// TwinCAT 3 PLC project AdsGamepad
// Title: AdsGamepad
// Company: Beckhoff Community
// Author: Beckhoff USA Community
// ProjectVersion: 2.3.0
// Description: A library to communicate with the ADS Gamepad Service
// ProgramVersion: 3.1.4026.24
// libraries:
//   Tc2_System, * (Beckhoff Automation GmbH)
//   Tc3_Module, * (Beckhoff Automation GmbH)
// project tree:
//   DUTs/ E_Gamepad_Battery_Levels.TcDUT, E_Gamepad_Battery_Types.TcDUT, E_Gamepad_Handshake_State.TcDUT, ST_Gamepad_ADS_Inputs.TcDUT, ST_Gamepad_Ext_ADS_Inputs.TcDUT, ST_Gamepad_Ext_Battery.TcDUT, ST_Gamepad_Ext_Buttons.TcDUT, ST_Gamepad_Motion.TcDUT, ST_Gamepad_Touch_Point.TcDUT, ST_Gamepad_Touchpad.TcDUT, ST_Gamepad_Buttons.TcDUT, ST_Gamepad_Command_Status.TcDUT, ST_Gamepad_DPad.TcDUT, ST_Gamepad_Joystick.TcDUT, ST_Gamepad_Rumble.TcDUT, ST_Gamepad_Service_Info.TcDUT, ST_Gamepad_Status.TcDUT
//   DUTs/LowerLevel/ ST_Gamepad_Buttons_Bits.TcDUT, ST_Gamepad_Ext_Touch_Raw.TcDUT, ST_Gamepad_State_Bits.TcDUT
//   FBs/ FB_Gamepad_Controller.TcPOU
//   Project Information/ F_GetCompany.TcPOU (not stored), F_GetTitle.TcPOU, F_GetVersion.TcPOU
//   Version/ Global_Version.TcGVL

// ---- DUTs/E_Gamepad_Battery_Levels.TcDUT
{attribute 'qualified_only'}
{attribute 'strict'}
TYPE E_Gamepad_Battery_Levels :
(
	// Battery is Empty or Unknown
	Empty := 0,
	// Battery is at low level
	Low := 1,
	// Battery is at medium level
	Medium := 2,
	// Battery is at full level
	Full := 3
);
END_TYPE

// ---- DUTs/E_Gamepad_Battery_Types.TcDUT
{attribute 'qualified_only'}
{attribute 'strict'}
TYPE E_Gamepad_Battery_Types :
(
	// Battery is disconnected
	Disconnected := 0,
	// Battery is wired
	Wired := 1,
	// Battery is alkaline
	Alkaline := 2,
	// Battery is NiMH
	NIMH := 3,
	// Battery is unknown
	Unknown := 4
);
END_TYPE

// ---- DUTs/E_Gamepad_Handshake_State.TcDUT
{attribute 'qualified_only'}
{attribute 'strict'}
TYPE E_Gamepad_Handshake_State :
(
	// No handshake attempt has run yet
	NotStarted := 0,
	// The read of the service info block is in flight
	Busy := 1,
	// The service answered and the contract versions are compatible
	Compatible := 2,
	// The last attempt got no answer. The service predates the info block or was not
	// reachable yet; the handshake keeps retrying. Data exchange still works
	Unsupported := 3,
	// The service speaks a newer contract major version. Check for a library update
	Mismatch := 4
);
END_TYPE

// ---- DUTs/LowerLevel/ST_Gamepad_Buttons_Bits.TcDUT
TYPE ST_Gamepad_Buttons_Bits :
STRUCT
	xDPAD_UP  			: BIT;
    xDPAD_DOWN  		: BIT;
    xDPAD_LEFT  		: BIT;
    xDPAD_RIGHT  		: BIT;
    xSTART  			: BIT;
    xBACK  				: BIT;
    xLEFT_THUMB  		: BIT;
    xRIGHT_THUMB  		: BIT;   
	xLEFT_SHOULDER  	: BIT;
    xRIGHT_SHOULDER  	: BIT;
	{attribute 'hide'}
	xFiller1 			: BIT;
	{attribute 'hide'}
	xFiller2			: BIT;
	xA  				: BIT;
	xB  				: BIT;
	xX  				: BIT;
	xY  				: BIT;
END_STRUCT
END_TYPE

// ---- DUTs/LowerLevel/ST_Gamepad_Ext_Touch_Raw.TcDUT
// One touchpad contact exactly as it arrives in the extended block.
// Use the P_Touchpad property for the friendly form. Layout is frozen.
{attribute 'pack_mode' := '4'}
TYPE ST_Gamepad_Ext_Touch_Raw :
STRUCT
	// 1 while a finger is on the pad, 0 otherwise
	nActive		: USINT;
	// Counts contacts, so a new touch gets a new number
	nContactId	: USINT;
	// Position across the pad, 0 to 1919
	nX			: UINT;
	// Position down the pad, 0 to 1079
	nY			: UINT;
END_STRUCT
END_TYPE

// ---- DUTs/LowerLevel/ST_Gamepad_State_Bits.TcDUT
TYPE ST_Gamepad_State_Bits :
STRUCT
	xConnected  				: BIT;
	xBattery_Type_Disconnected	: BIT;
	xBattery_Type_Wired			: BIT;
	xBattery_Type_Alkaline		: BIT;
	xBattery_Type_NIMH			: BIT;
	xBattery_Type_Unknown		: BIT;
	xBattery_Level_Empty		: BIT;
	xBattery_Level_Low			: BIT;
	xBattery_Level_Medium		: BIT;
	xBattery_Level_Full			: BIT;
	
	{attribute 'hide'}
	xFiller10					: BIT;
	{attribute 'hide'}
	xFiller11					: BIT;
	{attribute 'hide'}
	xFiller12					: BIT;
	{attribute 'hide'}
	xFiller13					: BIT;
	{attribute 'hide'}
	xFiller14					: BIT;
	{attribute 'hide'}
	xFiller15					: BIT;
END_STRUCT
END_TYPE

// ---- DUTs/ST_Gamepad_ADS_Inputs.TcDUT
TYPE ST_Gamepad_ADS_Inputs :
STRUCT
	// Controller Number
	iControllerNumber	: INT;
	// Struct of Left Joystick values
	stLeft_Joystick 	: ST_Gamepad_Joystick;
	// Struct of Right Joystick values
	stRight_Joystick 	: ST_Gamepad_Joystick;
	// Left Trigger value
	fLeft_Trigger 		: REAL;
	// Right Trigger value
	fRight_Trigger 		: REAL;
	// Struct of individual raw button bits read from the controller
	bButtons 			: ST_Gamepad_Buttons_Bits;
	// Struct of individual raw status bits read from the controller
	bStatus				: ST_Gamepad_State_Bits;
END_STRUCT
END_TYPE

// ---- DUTs/ST_Gamepad_Ext_ADS_Inputs.TcDUT
// Mirror of the 96 byte extended block served per controller since wire
// contract 1.3. Older services answer the read with an error and the
// struct then reads all zero. A slot without extended data, for example
// an Xbox controller, reads all zero with the present flag clear.
// Layout is frozen.
{attribute 'pack_mode' := '4'}
TYPE ST_Gamepad_Ext_ADS_Inputs :
STRUCT
	// Size of the block, 96 when the service serves it
	nExtSize			: UINT;
	// Layout version of the fields below, 1 today
	nExtLayoutVersion	: UINT;
	// Bit 0 PS, bit 1 Mute, bit 2 touchpad click
	nExtButtons			: WORD;
	// Bit 0 set means this slot supplies extended data right now.
	// Bit 1 set means the battery fields below hold data, since contract 1.4
	nExtFlags			: WORD;
	// Raw motion sensor values. Interpreting them is application code
	nGyroX				: INT;
	nGyroY				: INT;
	nGyroZ				: INT;
	nAccelX				: INT;
	nAccelY				: INT;
	nAccelZ				: INT;
	// Up to two touchpad contacts
	stTouch0			: ST_Gamepad_Ext_Touch_Raw;
	stTouch1			: ST_Gamepad_Ext_Touch_Raw;
	// Report counter from the pad, widened by the service. A value that
	// keeps moving proves the input stream is alive
	nSequence			: UDINT;
	// Battery data since contract 1.4, gated on flag bit 1: charge in
	// percent, then bit 0 charging and bit 1 full. Use P_Ext_Battery
	nBatteryPercent		: USINT;
	nBatteryFlags		: USINT;
	nReserved			: UINT;
	// Reserved for future contract versions, always zero today
	aReserved			: ARRAY [0..55] OF BYTE;
END_STRUCT
END_TYPE

// ---- DUTs/ST_Gamepad_Ext_Battery.TcDUT
// Battery state from the extended block. Valid only while bValid is TRUE:
// a service older than 2.6.0 does not serve it, an Xbox slot has none, and
// a pad error state reads as not valid rather than as a guess.
TYPE ST_Gamepad_Ext_Battery :
STRUCT
	// TRUE while the service supplies battery data for this slot
	bValid		: BOOL;
	// Charge from 0 to 100 percent
	nPercent	: USINT;
	// TRUE while the pad charges over its cable
	bCharging	: BOOL;
	// TRUE when the battery is full
	bFull		: BOOL;
END_STRUCT
END_TYPE

// ---- DUTs/ST_Gamepad_Ext_Buttons.TcDUT
// Buttons beyond the classic gamepad surface. A PlayStation pad supplies
// them through the extended block; on other pads they stay FALSE.
TYPE ST_Gamepad_Ext_Buttons :
STRUCT
	// The PS logo button
	bPS				: BOOL;
	// The microphone mute button
	bMute			: BOOL;
	// The touchpad pressed as a button
	bTouchpad_Click	: BOOL;
END_STRUCT
END_TYPE

// ---- DUTs/ST_Gamepad_Motion.TcDUT
// Raw motion sensor values from the pad. The units are the sensor's own;
// interpreting or filtering them is application code. At rest the gyro
// values show small noise and the accelerometer shows gravity.
TYPE ST_Gamepad_Motion :
STRUCT
	nGyroX	: INT;
	nGyroY	: INT;
	nGyroZ	: INT;
	nAccelX	: INT;
	nAccelY	: INT;
	nAccelZ	: INT;
END_STRUCT
END_TYPE

// ---- DUTs/ST_Gamepad_Touch_Point.TcDUT
// One finger on the touchpad in friendly form.
TYPE ST_Gamepad_Touch_Point :
STRUCT
	// TRUE while the finger touches the pad
	bActive		: BOOL;
	// Counts contacts, so a new touch gets a new number
	nContactId	: USINT;
	// Position across the pad, 0 to 1919
	nX			: UINT;
	// Position down the pad, 0 to 1079
	nY			: UINT;
END_STRUCT
END_TYPE

// ---- DUTs/ST_Gamepad_Touchpad.TcDUT
// The touchpad with its two possible contacts.
TYPE ST_Gamepad_Touchpad :
STRUCT
	stPoint1	: ST_Gamepad_Touch_Point;
	stPoint2	: ST_Gamepad_Touch_Point;
END_STRUCT
END_TYPE

// ---- DUTs/ST_Gamepad_Buttons.TcDUT
TYPE ST_Gamepad_Buttons :
STRUCT
	// Directional Pad Struct
	DPad				: ST_Gamepad_DPad;
	// Start Button
    bStart  			: BOOL;
	// Back Button
    bBack  				: BOOL;
	// Pressing in the Left Thumbstick
    bLeft_Thumbstick  	: BOOL;
	// Pressing in the Right Thumbstick
    bRight_Thumbstick  	: BOOL;
	// Left Shoulder Button  
	bLeft_Shoulder  	: BOOL;
	// Right Shoulder Button
    bRight_Shoulder  	: BOOL;
	// Button A
	bA_Button  			: BOOL;
	// Button B
	bB_Button  			: BOOL;
	// Button X
	bX_Button  			: BOOL;
	// Button Y
	bY_Button  			: BOOL;
END_STRUCT
END_TYPE

// ---- DUTs/ST_Gamepad_Command_Status.TcDUT
TYPE ST_Gamepad_Command_Status :
STRUCT
	// Command has been completed
	bDone 	: BOOL;
	// Command is busy
	bBusy 	: BOOL;
	// Command has an error
	bError 	: BOOL;
END_STRUCT
END_TYPE

// ---- DUTs/ST_Gamepad_DPad.TcDUT
TYPE ST_Gamepad_DPad :
STRUCT
	// Up Button on DPad
	bUp  		: BOOL;
	// Down Button on DPad
    bDown  		: BOOL;
	// Left Button on DPad
    bLeft  		: BOOL;
	// Right Button on DPad
    bRight  	: BOOL;
END_STRUCT
END_TYPE

// ---- DUTs/ST_Gamepad_Joystick.TcDUT
TYPE ST_Gamepad_Joystick :
STRUCT
	// Joystick's X Value (-100...100%)
	fX : REAL;
	// Joystick's Y Value (-100...100%)
	fY : REAL;
END_STRUCT
END_TYPE

// ---- DUTs/ST_Gamepad_Rumble.TcDUT
TYPE ST_Gamepad_Rumble :
STRUCT
	// Rumble of left motor (0..100%)
	fLeftMotor 	: REAL;
	// Rumble of right motor (0..100%)
	fRightMotor : REAL;
END_STRUCT
END_TYPE

// ---- DUTs/ST_Gamepad_Service_Info.TcDUT
// Mirror of the 32 byte service info block served at IndexGroup 16#F000.
// Services older than 2.1.0 do not serve this block. Layout is frozen.
TYPE ST_Gamepad_Service_Info :
STRUCT
	// Wire contract version the service speaks. This library expects major 1
	nContractMajor	: UINT;
	nContractMinor	: UINT;
	// Version of the running service program
	nServiceMajor	: UINT;
	nServiceMinor	: UINT;
	nServicePatch	: UINT;
	nReserved		: UINT;
	// Capability bits. Bit 0 means the XInput backend is present
	dwCapabilities	: UDINT;
	// Reserved for future contract versions, always zero today
	aReserved		: ARRAY [0..15] OF BYTE;
END_STRUCT
END_TYPE

// ---- DUTs/ST_Gamepad_Status.TcDUT
TYPE ST_Gamepad_Status :
STRUCT
	// Controller's ID
	iControllerNumber  	: INT;
	// Controller is connected to the PC
	bConnected  		: BOOL;
	// Controller is disconnected from the PC
	bDisconnected  		: BOOL;
	// Battery Type
	eBattery_Type 		: E_Gamepad_Battery_Types;
	// Battery Level
	eBattery_Level 		: E_Gamepad_Battery_Levels;
END_STRUCT
END_TYPE

// ---- Version/Global_Version.TcGVL
{attribute 'TcGenerated'}
{attribute 'no-analysis'}
{attribute 'linkalways'}
// This function has been automatically generated from the project information.
VAR_GLOBAL CONSTANT
	{attribute 'const_non_replaced'}
	stLibVersion_AdsGamepad : ST_LibVersion := (iMajor := 2, iMinor := 3, iBuild := 0, iRevision := 0, nFlags := 1, sVersion := '2.3.0');
END_VAR

// ---- FBs/FB_Gamepad_Controller.TcPOU
{attribute 'no_explicit_call' := 'do not call this FB directly, call Cycle instead'} 
FUNCTION_BLOCK FB_Gamepad_Controller
VAR
	{attribute 'hide'}
	_AmsNetId : T_AMSNETID;
	{attribute 'hide'}
	_WriteServerData : ADSWRITE;
	{attribute 'hide'}
	_ReadServerData : ADSREAD;
	// RAW ADS Inputs for debug (Use properties to access items)
	stGamepadInputs : ST_Gamepad_ADS_Inputs;
	{attribute 'hide'}
	_stRumble : ST_Gamepad_Rumble;
	{attribute 'hide'}
	_IDXGRP : UDINT;
	{attribute 'hide'}
	_rumbleCommand 			: ST_Gamepad_Command_Status;
	{attribute 'hide'}
	_stControllerButtons 	: ST_Gamepad_Buttons;
	{attribute 'hide'}
	_stControllerStatus		: ST_Gamepad_Status;
	{attribute 'hide'}
	_stLeftJoystick 		: ST_Gamepad_Joystick;
	{attribute 'hide'}
	_stRightJoystick 		: ST_Gamepad_Joystick;
	{attribute 'hide'}
	_fLeftTrigger 			: REAL;
	{attribute 'hide'}
	_fRightTrigger 			: REAL;
	{attribute 'hide'}
	_bSetRumbleEvent 		: BOOL; // Internal indication of an ADS write event
	{attribute 'hide'}
	_bSetRumbleEventLogged	: BOOL; // Check if the Set Rumble event is being called too many times
	{attribute 'hide'}
	_ReadServiceInfo : ADSREAD;
	{attribute 'hide'}
	_stServiceInfo : ST_Gamepad_Service_Info;
	{attribute 'hide'}
	_eHandshakeState : E_Gamepad_Handshake_State;
	{attribute 'hide'}
	_nHandshakeRetryCycles : UDINT; // Counts cycles between handshake retries after a failed attempt
	{attribute 'hide'}
	_ReadExtData : ADSREAD;
	// RAW extended block for debug (Use properties to access items)
	stGamepadExtInputs : ST_Gamepad_Ext_ADS_Inputs;
	{attribute 'hide'}
	_stExtButtons : ST_Gamepad_Ext_Buttons;
	{attribute 'hide'}
	_stTouchpad : ST_Gamepad_Touchpad;
	{attribute 'hide'}
	_stMotion : ST_Gamepad_Motion;
	{attribute 'hide'}
	_stExtBattery : ST_Gamepad_Ext_Battery;
END_VAR

// This method is called cyclically to update the controller inputs
METHOD Cycle : BOOL
// Read the current inputs
THIS^._ReadServerData(
	NETID:= THIS^._AmsNetId, 
	PORT:= 25733, 
	IDXGRP:= THIS^._IDXGRP, 
	IDXOFFS:= 0, 
	LEN:= SIZEOF(THIS^.stGamepadInputs), 
	DESTADDR:= ADR(THIS^.stGamepadInputs), 
	READ:= TRUE, 
	TMOUT:= T#5S,
	ERR=>);
	
// If there is an error in reading from the server, shut all inputs off
IF THIS^._ReadServerData.ERR THEN
	memset(ADR(THIS^.stGamepadInputs), 0, SIZEOF(THIS^.stGamepadInputs));
END_IF

// Stop read command
THIS^._ReadServerData(
	NETID:= THIS^._AmsNetId, 
	PORT:= 25733, 
	IDXGRP:= THIS^._IDXGRP, 
	IDXOFFS:= 0, 
	LEN:= SIZEOF(THIS^.stGamepadInputs), 
	DESTADDR:= ADR(THIS^.stGamepadInputs), 
	READ:= FALSE, 
	TMOUT:= T#5S,
	ERR=>);
	

// Handle any write requests for the rumble
// Write the new values
THIS^._WriteServerData(
	NETID:= THIS^._AmsNetId, 
	PORT:= 25733, 
	IDXGRP:= THIS^._IDXGRP, 
	IDXOFFS:= 16, 
	LEN:= SIZEOF(THIS^._stRumble), 
	SRCADDR:= ADR(THIS^._stRumble), 
	WRITE:= THIS^._bSetRumbleEvent, 
	TMOUT:= T#5S);
	
// Update the status of the current command if active
IF 	THIS^._bSetRumbleEvent THEN
	THIS^.P_SetRumble.bBusy := THIS^._WriteServerData.BUSY;
	THIS^.P_SetRumble.bError := THIS^._WriteServerData.ERR;
END_IF

// Check if it's done writing
IF THIS^._bSetRumbleEvent AND NOT THIS^._WriteServerData.BUSY THEN
	IF NOT THIS^._WriteServerData.ERR THEN
		THIS^.P_SetRumble.bDone := TRUE;
	END_IF
	// Turn off the write request
	THIS^._WriteServerData(
		NETID:= THIS^._AmsNetId, 
		PORT:= 25733, 
		IDXGRP:= THIS^._IDXGRP, 
		IDXOFFS:= 16, 
		LEN:= SIZEOF(THIS^._stRumble), 
		SRCADDR:= ADR(THIS^._stRumble), 
		WRITE:= FALSE, 
		TMOUT:= T#5S);

	THIS^._bSetRumbleEvent := FALSE;
END_IF

// Version handshake against the service info block at IndexGroup 16#F000.
// Services older than 2.1.0 answer with an error, which is fine. Data exchange works either way.
// A failed attempt reports Unsupported and retries in the background, so a service that starts
// after the PLC, for example right after an install, still gets a handshake without a PLC restart
CASE THIS^._eHandshakeState OF
	E_Gamepad_Handshake_State.NotStarted:
		THIS^._ReadServiceInfo(
			NETID:= THIS^._AmsNetId,
			PORT:= 25733,
			IDXGRP:= 16#F000,
			IDXOFFS:= 0,
			LEN:= SIZEOF(THIS^._stServiceInfo),
			DESTADDR:= ADR(THIS^._stServiceInfo),
			READ:= TRUE,
			TMOUT:= T#5S);
		THIS^._eHandshakeState := E_Gamepad_Handshake_State.Busy;

	E_Gamepad_Handshake_State.Busy:
		THIS^._ReadServiceInfo(READ:= TRUE);
		IF THIS^._ReadServiceInfo.ERR THEN
			// No answer. The service predates version 2.1.0 or it was not reachable, for example
			// while it was still starting. The Unsupported case below retries later
			memset(ADR(THIS^._stServiceInfo), 0, SIZEOF(THIS^._stServiceInfo));
			THIS^._eHandshakeState := E_Gamepad_Handshake_State.Unsupported;
			THIS^._ReadServiceInfo(READ:= FALSE);
		ELSIF NOT THIS^._ReadServiceInfo.BUSY THEN
			IF THIS^._stServiceInfo.nContractMajor = 1 THEN
				THIS^._eHandshakeState := E_Gamepad_Handshake_State.Compatible;
			ELSE
				ADSLOGSTR( msgCtrlMask := ADSLOG_MSGTYPE_WARN, msgFmtStr := 'PLC Msg.: The ADS Gamepad Service speaks a newer wire contract, update the AdsGamepad library: %s', strArg := 'FB_Gamepad_Controller');
				THIS^._eHandshakeState := E_Gamepad_Handshake_State.Mismatch;
			END_IF
			THIS^._ReadServiceInfo(READ:= FALSE);
		END_IF

	E_Gamepad_Handshake_State.Unsupported:
		// Retry the handshake in the background without leaving the reported state,
		// so consumers watching P_Handshake_State never see it flap. A genuinely old
		// service answers every retry with an error and the state simply stays
		// Unsupported; a service that was only starting late answers and the state
		// moves on. 5000 cycles is five seconds at a one millisecond PLC cycle
		THIS^._nHandshakeRetryCycles := THIS^._nHandshakeRetryCycles + 1;
		IF THIS^._nHandshakeRetryCycles >= 5000 THEN
			THIS^._ReadServiceInfo(
				NETID:= THIS^._AmsNetId,
				PORT:= 25733,
				IDXGRP:= 16#F000,
				IDXOFFS:= 0,
				LEN:= SIZEOF(THIS^._stServiceInfo),
				DESTADDR:= ADR(THIS^._stServiceInfo),
				READ:= TRUE,
				TMOUT:= T#5S);
			IF THIS^._ReadServiceInfo.ERR THEN
				// Still no answer; reset the read and count up to the next attempt
				memset(ADR(THIS^._stServiceInfo), 0, SIZEOF(THIS^._stServiceInfo));
				THIS^._ReadServiceInfo(READ:= FALSE);
				THIS^._nHandshakeRetryCycles := 0;
			ELSIF NOT THIS^._ReadServiceInfo.BUSY THEN
				IF THIS^._stServiceInfo.nContractMajor = 1 THEN
					THIS^._eHandshakeState := E_Gamepad_Handshake_State.Compatible;
				ELSE
					ADSLOGSTR( msgCtrlMask := ADSLOG_MSGTYPE_WARN, msgFmtStr := 'PLC Msg.: The ADS Gamepad Service speaks a newer wire contract, update the AdsGamepad library: %s', strArg := 'FB_Gamepad_Controller');
					THIS^._eHandshakeState := E_Gamepad_Handshake_State.Mismatch;
				END_IF
				THIS^._ReadServiceInfo(READ:= FALSE);
				THIS^._nHandshakeRetryCycles := 0;
			END_IF
		END_IF
END_CASE
END_METHOD

METHOD FB_init : BOOL
VAR_INPUT
	bInitRetains : BOOL; // if TRUE, the retain variables are initialized (warm start / cold start)
	bInCopyCode : BOOL;  // if TRUE, the instance afterwards gets moved into the copy code (online change)
	NetID 				: T_AMSNETID := ''; // AMS Net ID of the ADS Gamepad Service
	iControllerNumber 	: UINT(1..4) := 1; // The controller number for the controller you'd like to use
END_VAR
THIS^._AmsNetId := NetID;
THIS^._IDXGRP := iControllerNumber * 16#10000;
END_METHOD

{attribute 'monitoring':='call'}
// Structure of the different active buttons
PROPERTY P_Buttons : REFERENCE TO ST_Gamepad_Buttons
GET
IF THIS^.stGamepadInputs.bStatus.xConnected THEN	
	THIS^._stControllerButtons.DPad.bUp				:= THIS^.stGamepadInputs.bButtons.xDPAD_UP;
	THIS^._stControllerButtons.DPad.bDown			:= THIS^.stGamepadInputs.bButtons.xDPAD_DOWN;
	THIS^._stControllerButtons.DPad.bLeft			:= THIS^.stGamepadInputs.bButtons.xDPAD_LEFT;
	THIS^._stControllerButtons.DPad.bRight			:= THIS^.stGamepadInputs.bButtons.xDPAD_RIGHT;
	THIS^._stControllerButtons.bStart  				:= THIS^.stGamepadInputs.bButtons.xSTART;
	THIS^._stControllerButtons.bBack  				:= THIS^.stGamepadInputs.bButtons.xBACK;
	THIS^._stControllerButtons.bLeft_Thumbstick  	:= THIS^.stGamepadInputs.bButtons.xLEFT_THUMB;
	THIS^._stControllerButtons.bRight_Thumbstick 	:= THIS^.stGamepadInputs.bButtons.xRIGHT_THUMB;
	THIS^._stControllerButtons.bLeft_Shoulder  		:= THIS^.stGamepadInputs.bButtons.xLEFT_SHOULDER;
	THIS^._stControllerButtons.bRight_Shoulder  	:= THIS^.stGamepadInputs.bButtons.xRIGHT_SHOULDER;
	THIS^._stControllerButtons.bA_Button  			:= THIS^.stGamepadInputs.bButtons.xA;
	THIS^._stControllerButtons.bB_Button  			:= THIS^.stGamepadInputs.bButtons.xB;
	THIS^._stControllerButtons.bX_Button  			:= THIS^.stGamepadInputs.bButtons.xX;
	THIS^._stControllerButtons.bY_Button  			:= THIS^.stGamepadInputs.bButtons.xY;
ELSE
	THIS^._stControllerButtons.DPad.bUp				:= FALSE;
	THIS^._stControllerButtons.DPad.bDown			:= FALSE;
	THIS^._stControllerButtons.DPad.bLeft			:= FALSE;
	THIS^._stControllerButtons.DPad.bRight			:= FALSE;
	THIS^._stControllerButtons.bStart  				:= FALSE;
	THIS^._stControllerButtons.bBack  				:= FALSE;
	THIS^._stControllerButtons.bLeft_Thumbstick  	:= FALSE;
	THIS^._stControllerButtons.bRight_Thumbstick 	:= FALSE;
	THIS^._stControllerButtons.bLeft_Shoulder  		:= FALSE;
	THIS^._stControllerButtons.bRight_Shoulder  	:= FALSE;
	THIS^._stControllerButtons.bA_Button  			:= FALSE;
	THIS^._stControllerButtons.bB_Button  			:= FALSE;
	THIS^._stControllerButtons.bX_Button  			:= FALSE;
	THIS^._stControllerButtons.bY_Button  			:= FALSE;
END_IF
P_Buttons REF= THIS^._stControllerButtons;
END_GET
END_PROPERTY

{attribute 'monitoring':='call'}
// Returns a structure of data for the XY Joystick values
PROPERTY P_Left_Joystick : REFERENCE TO ST_Gamepad_Joystick
GET
IF THIS^.stGamepadInputs.bStatus.xConnected THEN	
	THIS^._stLeftJoystick.fX := THIS^.stGamepadInputs.stLeft_Joystick.fX;
	THIS^._stLeftJoystick.fY := THIS^.stGamepadInputs.stLeft_Joystick.fY;
ELSE
	THIS^._stLeftJoystick.fX := 0;
	THIS^._stLeftJoystick.fY := 0;
END_IF
P_Left_Joystick REF= THIS^._stLeftJoystick;
END_GET
END_PROPERTY

{attribute 'monitoring':='call'}
// Left trigger value
PROPERTY P_Left_Trigger : REFERENCE TO REAL
GET
IF THIS^.stGamepadInputs.bStatus.xConnected THEN	
	THIS^._fLeftTrigger := THIS^.stGamepadInputs.fLeft_Trigger;
ELSE
	THIS^._fLeftTrigger := 0;
END_IF
P_Left_Trigger REF= THIS^._fLeftTrigger;
END_GET
END_PROPERTY

{attribute 'monitoring':='call'}
// Returns a structure of data for the XY Joystick values
PROPERTY P_Right_Joystick : REFERENCE TO ST_Gamepad_Joystick
GET
IF THIS^.stGamepadInputs.bStatus.xConnected THEN	
	THIS^._stRightJoystick.fX := THIS^.stGamepadInputs.stRight_Joystick.fX;
	THIS^._stRightJoystick.fY := THIS^.stGamepadInputs.stRight_Joystick.fY;
ELSE
	THIS^._stRightJoystick.fX := 0;
	THIS^._stRightJoystick.fY := 0;
END_IF
P_Right_Joystick REF= THIS^._stRightJoystick;
END_GET
END_PROPERTY

{attribute 'monitoring':='call'}
// Right trigger value
PROPERTY P_Right_Trigger : REFERENCE TO REAL
GET
IF THIS^.stGamepadInputs.bStatus.xConnected THEN	
	THIS^._fRightTrigger := THIS^.stGamepadInputs.fRight_Trigger;
ELSE
	THIS^._fRightTrigger := 0;
END_IF
P_Right_Trigger REF= THIS^._fRightTrigger;
END_GET
END_PROPERTY

{attribute 'monitoring':='call'}
// Status of the SetRumble method
PROPERTY P_SetRumble : REFERENCE TO ST_Gamepad_Command_Status
GET
P_SetRumble REF= THIS^._rumbleCommand;
END_GET
END_PROPERTY

{attribute 'monitoring':='call'}
// Structure of the controller capabilites and status
PROPERTY P_Status : REFERENCE TO ST_Gamepad_Status
GET
IF THIS^.stGamepadInputs.bStatus.xConnected THEN	
	THIS^._stControllerStatus.bConnected 		:= TRUE;
	THIS^._stControllerStatus.bDisconnected 	:= FALSE;
	THIS^._stControllerStatus.iControllerNumber := THIS^.stGamepadInputs.iControllerNumber;
ELSE
	THIS^._stControllerStatus.bConnected 		:= FALSE;
	THIS^._stControllerStatus.bDisconnected 	:= TRUE;
	THIS^._stControllerStatus.iControllerNumber := 0;
END_IF

IF THIS^.stGamepadInputs.bStatus.xBattery_Type_Disconnected THEN
	THIS^._stControllerStatus.eBattery_Type := E_Gamepad_Battery_Types.Disconnected;
END_IF

IF THIS^.stGamepadInputs.bStatus.xBattery_Type_Wired THEN
	THIS^._stControllerStatus.eBattery_Type := E_Gamepad_Battery_Types.Wired;
END_IF

IF THIS^.stGamepadInputs.bStatus.xBattery_Type_Alkaline THEN
	THIS^._stControllerStatus.eBattery_Type := E_Gamepad_Battery_Types.Alkaline;
END_IF

IF THIS^.stGamepadInputs.bStatus.xBattery_Type_NIMH THEN
	THIS^._stControllerStatus.eBattery_Type := E_Gamepad_Battery_Types.NIMH;
END_IF

IF THIS^.stGamepadInputs.bStatus.xBattery_Type_Unknown THEN
	THIS^._stControllerStatus.eBattery_Type := E_Gamepad_Battery_Types.Unknown;
END_IF

IF THIS^.stGamepadInputs.bStatus.xBattery_Level_Empty THEN
	THIS^._stControllerStatus.eBattery_Level := E_Gamepad_Battery_Levels.Empty;
END_IF

IF THIS^.stGamepadInputs.bStatus.xBattery_Level_Low THEN
	THIS^._stControllerStatus.eBattery_Level := E_Gamepad_Battery_Levels.Low;
END_IF

IF THIS^.stGamepadInputs.bStatus.xBattery_Level_Medium THEN
	THIS^._stControllerStatus.eBattery_Level := E_Gamepad_Battery_Levels.Medium;
END_IF

IF THIS^.stGamepadInputs.bStatus.xBattery_Level_Full THEN
	THIS^._stControllerStatus.eBattery_Level := E_Gamepad_Battery_Levels.Full;
END_IF


P_Status REF= THIS^._stControllerStatus;
END_GET
END_PROPERTY

{attribute 'monitoring':='call'}
// Result of the version handshake with the service. Unsupported retries in the background
PROPERTY P_Handshake_State : E_Gamepad_Handshake_State
GET
P_Handshake_State := THIS^._eHandshakeState;
END_GET
END_PROPERTY

{attribute 'monitoring':='call'}
// Version and capability info read from the service during the handshake
PROPERTY P_Service_Info : REFERENCE TO ST_Gamepad_Service_Info
GET
P_Service_Info REF= THIS^._stServiceInfo;
END_GET
END_PROPERTY

// Sets the rumble for the controller
METHOD SetRumble : BOOL
VAR_INPUT
	// Left motor speed (0..100%)
	fLeftMotor : REAL;
	// Right motor speed (0..100%)
	fRightMotor : REAL;
END_VAR
// When the method is called, check if a write is in progress
IF THIS^._bSetRumbleEvent THEN
	// ADS you are doing that too much
	IF NOT THIS^._bSetRumbleEventLogged THEN
		ADSLOGSTR( msgCtrlMask := ADSLOG_MSGTYPE_WARN, msgFmtStr := 'PLC Msg.: Command being called too often, wait for done bit: %s', strArg := 'SetRumble()');
		THIS^._bSetRumbleEventLogged := TRUE;
	END_IF	
ELSE
	// Check if the value is within range
	IF fLeftMotor > 100 THEN
		THIS^._stRumble.fLeftMotor := 100.0;
	ELSIF fLeftMotor < 0 THEN
		THIS^._stRumble.fLeftMotor := 0.0;
	ELSE
		THIS^._stRumble.fLeftMotor := fLeftMotor;
	END_IF
	
	// Check if the value is within range
	IF fRightMotor > 100 THEN
		THIS^._stRumble.fRightMotor := 100.0;
	ELSIF fRightMotor < 0 THEN
		THIS^._stRumble.fRightMotor := 0.0;
	ELSE
		THIS^._stRumble.fRightMotor := fRightMotor;
	END_IF
	
	//Reset all status for the command
	THIS^.P_SetRumble.bDone := FALSE;
	THIS^.P_SetRumble.bBusy := FALSE;
	THIS^.P_SetRumble.bError := FALSE;

	// Set the high bit on the write command
	THIS^._bSetRumbleEvent := TRUE;
END_IF

// If it's done, set the current even in progress to false
IF P_SetRumble.bDone THEN
	THIS^._bSetRumbleEvent := FALSE;
END_IF

// Event Received
SetRumble := THIS^._bSetRumbleEvent;
END_METHOD

// Reads the 96 byte extended block, wire contract 1.3. Call this once per
// PLC cycle in addition to Cycle when the extended data is wanted; it costs
// one extra ADS read per cycle and programs that never call it behave
// exactly as before. A service older than 2.5.0 answers with an error and
// the block then reads all zero, the same fail safe as everywhere else.
METHOD ReadExtended : BOOL
// Read the current extended block
THIS^._ReadExtData(
	NETID:= THIS^._AmsNetId,
	PORT:= 25733,
	IDXGRP:= THIS^._IDXGRP + 16#100,
	IDXOFFS:= 0,
	LEN:= SIZEOF(THIS^.stGamepadExtInputs),
	DESTADDR:= ADR(THIS^.stGamepadExtInputs),
	READ:= TRUE,
	TMOUT:= T#5S,
	ERR=>);

// If there is an error in reading from the server, shut all values off
IF THIS^._ReadExtData.ERR THEN
	memset(ADR(THIS^.stGamepadExtInputs), 0, SIZEOF(THIS^.stGamepadExtInputs));
END_IF

// Stop read command
THIS^._ReadExtData(
	NETID:= THIS^._AmsNetId,
	PORT:= 25733,
	IDXGRP:= THIS^._IDXGRP + 16#100,
	IDXOFFS:= 0,
	LEN:= SIZEOF(THIS^.stGamepadExtInputs),
	DESTADDR:= ADR(THIS^.stGamepadExtInputs),
	READ:= FALSE,
	TMOUT:= T#5S,
	ERR=>);
END_METHOD

{attribute 'monitoring':='call'}
// Buttons beyond the classic surface, from the extended block
PROPERTY P_Ext_Buttons : REFERENCE TO ST_Gamepad_Ext_Buttons
GET
IF (THIS^.stGamepadExtInputs.nExtFlags AND 16#0001) <> 0 THEN
	THIS^._stExtButtons.bPS 			:= (THIS^.stGamepadExtInputs.nExtButtons AND 16#0001) <> 0;
	THIS^._stExtButtons.bMute 			:= (THIS^.stGamepadExtInputs.nExtButtons AND 16#0002) <> 0;
	THIS^._stExtButtons.bTouchpad_Click := (THIS^.stGamepadExtInputs.nExtButtons AND 16#0004) <> 0;
ELSE
	THIS^._stExtButtons.bPS 			:= FALSE;
	THIS^._stExtButtons.bMute 			:= FALSE;
	THIS^._stExtButtons.bTouchpad_Click := FALSE;
END_IF
P_Ext_Buttons REF= THIS^._stExtButtons;
END_GET
END_PROPERTY

{attribute 'monitoring':='call'}
// The two touchpad contacts from the extended block
PROPERTY P_Touchpad : REFERENCE TO ST_Gamepad_Touchpad
GET
IF (THIS^.stGamepadExtInputs.nExtFlags AND 16#0001) <> 0 THEN
	THIS^._stTouchpad.stPoint1.bActive 		:= THIS^.stGamepadExtInputs.stTouch0.nActive <> 0;
	THIS^._stTouchpad.stPoint1.nContactId 	:= THIS^.stGamepadExtInputs.stTouch0.nContactId;
	THIS^._stTouchpad.stPoint1.nX 			:= THIS^.stGamepadExtInputs.stTouch0.nX;
	THIS^._stTouchpad.stPoint1.nY 			:= THIS^.stGamepadExtInputs.stTouch0.nY;
	THIS^._stTouchpad.stPoint2.bActive 		:= THIS^.stGamepadExtInputs.stTouch1.nActive <> 0;
	THIS^._stTouchpad.stPoint2.nContactId 	:= THIS^.stGamepadExtInputs.stTouch1.nContactId;
	THIS^._stTouchpad.stPoint2.nX 			:= THIS^.stGamepadExtInputs.stTouch1.nX;
	THIS^._stTouchpad.stPoint2.nY 			:= THIS^.stGamepadExtInputs.stTouch1.nY;
ELSE
	memset(ADR(THIS^._stTouchpad), 0, SIZEOF(THIS^._stTouchpad));
END_IF
P_Touchpad REF= THIS^._stTouchpad;
END_GET
END_PROPERTY

{attribute 'monitoring':='call'}
// Raw motion sensor values from the extended block
PROPERTY P_Motion : REFERENCE TO ST_Gamepad_Motion
GET
IF (THIS^.stGamepadExtInputs.nExtFlags AND 16#0001) <> 0 THEN
	THIS^._stMotion.nGyroX 	:= THIS^.stGamepadExtInputs.nGyroX;
	THIS^._stMotion.nGyroY 	:= THIS^.stGamepadExtInputs.nGyroY;
	THIS^._stMotion.nGyroZ 	:= THIS^.stGamepadExtInputs.nGyroZ;
	THIS^._stMotion.nAccelX := THIS^.stGamepadExtInputs.nAccelX;
	THIS^._stMotion.nAccelY := THIS^.stGamepadExtInputs.nAccelY;
	THIS^._stMotion.nAccelZ := THIS^.stGamepadExtInputs.nAccelZ;
ELSE
	memset(ADR(THIS^._stMotion), 0, SIZEOF(THIS^._stMotion));
END_IF
P_Motion REF= THIS^._stMotion;
END_GET
END_PROPERTY

{attribute 'monitoring':='call'}
// Battery state from the extended block, valid while bValid is TRUE
PROPERTY P_Ext_Battery : REFERENCE TO ST_Gamepad_Ext_Battery
GET
IF (THIS^.stGamepadExtInputs.nExtFlags AND 16#0002) <> 0 THEN
	THIS^._stExtBattery.bValid 		:= TRUE;
	THIS^._stExtBattery.nPercent 	:= THIS^.stGamepadExtInputs.nBatteryPercent;
	THIS^._stExtBattery.bCharging 	:= (THIS^.stGamepadExtInputs.nBatteryFlags AND 16#01) <> 0;
	THIS^._stExtBattery.bFull 		:= (THIS^.stGamepadExtInputs.nBatteryFlags AND 16#02) <> 0;
ELSE
	THIS^._stExtBattery.bValid 		:= FALSE;
	THIS^._stExtBattery.nPercent 	:= 0;
	THIS^._stExtBattery.bCharging 	:= FALSE;
	THIS^._stExtBattery.bFull 		:= FALSE;
END_IF
P_Ext_Battery REF= THIS^._stExtBattery;
END_GET
END_PROPERTY

{attribute 'monitoring':='call'}
// Report counter from the extended block. A value that keeps moving proves
// the input stream is alive; a program can watchdog it
PROPERTY P_Sequence : UDINT
GET
P_Sequence := THIS^.stGamepadExtInputs.nSequence;
END_GET
END_PROPERTY

END_FUNCTION_BLOCK

// ---- Project Information/F_GetTitle.TcPOU
// This function has been automatically generated from the project information.
{attribute 'signature_flag' := '1073741824'}
{attribute 'TcGenerated'}
{attribute 'no-analysis'}
FUNCTION F_GetTitle : WSTRING
VAR_INPUT
	
END_VAR

F_GetTitle := "AdsGamepad";

END_FUNCTION

// ---- Project Information/F_GetVersion.TcPOU
// This function has been automatically generated from the project information.
{attribute 'signature_flag' := '1073741824'}
{attribute 'TcGenerated'}
{attribute 'no-analysis'}
FUNCTION F_GetVersion : ST_LibVersion
VAR_INPUT
	
END_VAR

F_GetVersion.iMajor := 2;
F_GetVersion.iMinor := 3;
F_GetVersion.iBuild := 0;
F_GetVersion.iRevision := 0;
F_GetVersion.sVersion := '2.3.0';
F_GetVersion.nFlags := 1;

END_FUNCTION
